// TwinCAT 3 PLC project IO_Link
// Title: ZigaLibs.IoLink
// Company: Ziga Javornik
// Author: Ziga Javornik
// ProjectVersion: 0.0.0.1
// Description: IO link implementaiton libray
// ProgramVersion: 3.1.4026.26
// libraries:
//   Tc2_Standard, * (Beckhoff Automation GmbH)
//   Tc2_System, * (Beckhoff Automation GmbH)
//   Tc3_Module, * (Beckhoff Automation GmbH)
//   TcUnit, * (www.tcunit.org)
//   ZigaLibs.Logging, * (Ziga Javornik)
// project tree:
//   SOURCE/ FB_IoLinkChannel_64Byte.TcPOU, FB_IoLinkState.TcPOU, ST_IoLink_ChannelState.TcDUT, T_IoLink64ByteData.TcDUT
//   TESTS/ PRG_TESTS.TcPOU (not stored)
//   TESTS/Test suites/ FB_SUT_Tests.TcPOU (not stored)
// (motion and I/O tree: see PLC project logging)
// real-time tasks:
//   TASK TestsTask: cycle T#10ms, priority 20, ADS port 350
//   TASK PlcTask: cycle T#10ms, priority 21, ADS port 351

// ---- SOURCE/ST_IoLink_ChannelState.TcDUT
{attribute 'qualified_only'}
{attribute 'strict'}
{attribute 'to_string'}
TYPE ST_IoLink_ChannelState :
STRUCT
	PortDisabled 				: BOOL;
	PortInStdDigIn 				: BOOL;
	PortInStdDigOut				: BOOL;
	PortInCommunicationOP		: BOOL;
	PortInCommunicationCOMSTOP	: BOOL;
	WatchdogDetected			: BOOL;
	InternalError				: BOOL;
	InvalidDeviceId				: BOOL;
	InvalidVendorId				: BOOL;
	InvalidIoLinkVersion		: BOOL;
	InvalidFrameCapability		: BOOL;
	InvalidCycleTime			: BOOL;
	InvalidPD_InLength			: BOOL;
	InvalidPD_OutLength			: BOOL;
	NoDeviceDetected			: BOOL;
	ErrorPreoperate				: BOOL;
END_STRUCT
END_TYPE

// ---- SOURCE/T_IoLink64ByteData.TcDUT
TYPE 
	T_IoLink64ByteData : ARRAY[0..7] OF BYTE; 
END_TYPE

// ---- SOURCE/FB_IoLinkChannel_64Byte.TcPOU
FUNCTION_BLOCK ABSTRACT FB_IoLinkChannel_64Byte
VAR_INPUT
END_VAR
VAR_OUTPUT
END_VAR
VAR
	Inputs 	AT %I*	: T_IoLink64ByteData;
	Outputs	AT %Q*	: T_IoLink64ByteData;
END_VAR

END_FUNCTION_BLOCK

// ---- SOURCE/FB_IoLinkState.TcPOU
FUNCTION_BLOCK ABSTRACT FB_IoLinkState
VAR_INPUT
END_VAR
VAR_OUTPUT
END_VAR
VAR
	State	 AT%I*	: USINT;
	_channelState 	: ST_IoLink_ChannelState;
	_logger			: REFERENCE TO ZigaLibs_Logging.I_Logger;
END_VAR

 {attribute 'monitoring' := 'variable'}
// Gets the IO link channel state info
PROPERTY PUBLIC ChannelState : REFERENCE TO ST_IoLink_ChannelState
GET
_channelState := THIS^.GetChannelState();
ChannelState REF= _channelState;
END_GET
END_PROPERTY

METHOD FB_init : BOOL
VAR_INPUT
	bInitRetains : BOOL; // if TRUE, the retain variables are initialized (warm start / cold start)
	bInCopyCode : BOOL;  // if TRUE, the instance afterwards gets moved into the copy code (online change)
	logger			: REFERENCE TO ZigaLibs_Logging.I_Logger;
END_VAR
_logger REF= logger;
END_METHOD

// Gets the channel state based on the State value transfered from the hardware device
METHOD PUBLIC GetChannelState : ST_IoLink_ChannelState

VAR
	nMaskedState	: USINT;
	result			: ST_IoLink_ChannelState;
END_VAR
nMaskedState := 16#0F AND THIS^.State;
result.PortDisabled := nMaskedState = 16#00;
result.PortInStdDigIn := nMaskedState = 16#01;
result.PortInStdDigOut := nMaskedState = 16#02;
result.PortInCommunicationOP := nMaskedState = 16#03;
result.PortInCommunicationCOMSTOP := nMaskedState = 16#04;

nMaskedState := 16#F0 AND THIS^.State;
result.WatchdogDetected := nMaskedState = 16#10;
result.InternalError := nMaskedState = 16#20;
result.InvalidDeviceId := nMaskedState = 16#30;
result.InvalidVendorId := nMaskedState = 16#40;
result.InvalidIoLinkVersion := nMaskedState = 16#50;
result.InvalidFrameCapability := nMaskedState = 16#60;
result.InvalidCycleTime := nMaskedState = 16#70;
result.InvalidPD_InLength := nMaskedState = 16#80;
result.InvalidPD_OutLength := nMaskedState = 16#90;
result.NoDeviceDetected := nMaskedState = 16#A0;
result.ErrorPreoperate := nMaskedState = 16#B0;

GetChannelState := result;
END_METHOD

END_FUNCTION_BLOCK
